TYPE SequenceCommand :
STRUCT
	Start : PLCopenCommand;
	Stop : PLCopenCommand;
END_STRUCT
END_TYPE

(* stored: Version 1.1.0.1
   DUT SequenceCommand: Id {5f5128e9-4988-0cd7-37c1-c51312994c6b} *)
